PROGRAM PRG_EtherCATSimMasterDiag
VAR
	EcSimNetorkDiag		AT%I* 	:ARRAY[1..NumOfEcSimNetWorks] OF ST_EC_SIM_Device_Inputs;
	EcDevState					:ARRAY[1..NumOfEcSimNetWorks] OF STRING;
END_VAR
VAR CONSTANT
	NumOfEcSimNetWorks			:UDINT:=6;
END_VAR
VAR_TEMP
	i							:UDINT;
END_VAR


FOR i:=1 TO NumOfEcSimNetWorks DO
	EcDevState[i]:=F_ConvMasterDevStateToString(nState:=EcSimNetorkDiag[i].DevState);
END_FOR

END_PROGRAM

(* stored: Version 1.1.0.1, ProductVersion 3.1.4024.11
   POU PRG_EtherCATSimMasterDiag: Id {ae80a5f1-ab9e-463d-a30e-c2f6f38f86cf}, SpecialFunc None *)
